// TIA Portal V17 export
// export: Created 2021-09-22T08:50:40.0817292Z, ExportSetting WithDefaults, DisplayName Totally Integrated Automation Portal, DisplayVersion V17, DisplayName TIA Portal Openness, DisplayVersion V17, DisplayName TIA Portal Version Control Interface, DisplayVersion V17, DisplayName SINAMICS Startdrive Advanced, DisplayVersion V17, DisplayName SINAMICS Startdrive G130, G150, S120, S150, SINAMICS MV, S210, DisplayVersion V17, DisplayName SINAMICS Startdrive G110M, G120, G120C, G120D, G120P, G115D, DisplayVersion V17, DisplayName STEP 7 Professional, DisplayVersion V17, DisplayName STEP 7 Safety, DisplayVersion V17, DisplayName WinCC Advanced / Unified PC, DisplayVersion V17
FUNCTION_BLOCK "MainProgram"   // FB1, LAD
{ S7_Optimized_Access := 'TRUE' }
VERSION : 0.1
// stored: AutoNumber true, IsIECCheckEnabled false, IsRetainMemResEnabled false, MemoryReserve 100, SetENOAutomatically false, UDAEnableTagReadback false
   VAR_IN_OUT
      Hmi : "Visu_type";
   END_VAR
   VAR
      MotorCem : "MotorCem_type";
      Motor { S7_SetPoint := 'True'} : Array[0.."MAX_MOTOR_IDX"] of "Motor_type";
      Visu_0 { S7_SetPoint := 'True'} : "Visu";
   END_VAR
BEGIN

REGION Network 1
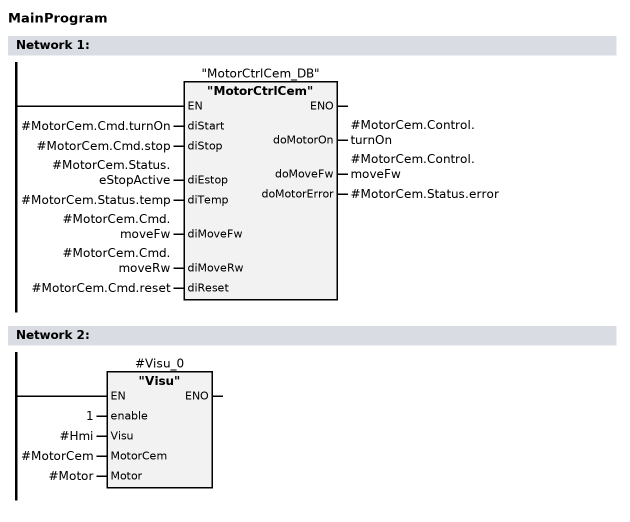
   RUNG wire#powerrail
      "MotorCtrlCem_DB"(diStart := #MotorCem.Cmd.turnOn, diStop := #MotorCem.Cmd.stop, diEstop := #MotorCem.Status.eStopActive, diTemp := #MotorCem.Status.temp, diMoveFw := #MotorCem.Cmd.moveFw, diMoveRw := #MotorCem.Cmd.moveRw, diReset := #MotorCem.Cmd.reset, doMotorOn => #MotorCem.Control.turnOn, doMoveFw => #MotorCem.Control.moveFw, doMotorError => #MotorCem.Status.error)
   END_RUNG
   // the same network as SCL:
   "MotorCtrlCem_DB"(diStart := #MotorCem.Cmd.turnOn,   // "MotorCtrlCem"
                     diStop := #MotorCem.Cmd.stop,
                     diEstop := #MotorCem.Status.eStopActive,
                     diTemp := #MotorCem.Status.temp,
                     diMoveFw := #MotorCem.Cmd.moveFw,
                     diMoveRw := #MotorCem.Cmd.moveRw,
                     diReset := #MotorCem.Cmd.reset,
                     doMotorOn => #MotorCem.Control.turnOn,
                     doMoveFw => #MotorCem.Control.moveFw,
                     doMotorError => #MotorCem.Status.error);
END_REGION

REGION Network 2
   RUNG wire#powerrail
      #Visu_0(enable := 1, Visu := #Hmi, MotorCem := #MotorCem, Motor := #Motor)
   END_RUNG
   // the same network as SCL:
   #Visu_0(enable := 1, Visu := #Hmi, MotorCem := #MotorCem, Motor := #Motor);   // "Visu"
END_REGION
END_FUNCTION_BLOCK
